(* IEC 61131-3 sources: kerf/packages/kerf-plc/tests/fixtures, 2 files *)

(* ---- blinker.st ---- *)
(* Blinker POU — drives pulse_out at 1 Hz using a TON timer *)
FUNCTION_BLOCK Blinker
VAR
    clock_in : BOOL;
    pulse_out : BOOL;
    t : TON;
END_VAR

(* Update the on-delay timer *)
t(IN := clock_in, PT := T#1s);

(* Latch output from timer Q output *)
pulse_out := t.Q;

END_FUNCTION_BLOCK

(* ---- conveyor.st ---- *)
(* Conveyor POU — start/stop/e-stop control with motor output *)
FUNCTION_BLOCK Conveyor
VAR_INPUT
    start_btn  : BOOL;
    stop_btn   : BOOL;
    estop      : BOOL;
END_VAR
VAR_OUTPUT
    motor_run  : BOOL;
    fault_lamp : BOOL;
END_VAR
VAR
    running    : BOOL;
END_VAR

(* Emergency stop overrides everything *)
IF estop THEN
    running    := FALSE;
    fault_lamp := TRUE;
ELSIF start_btn AND NOT stop_btn THEN
    running    := TRUE;
    fault_lamp := FALSE;
ELSIF stop_btn THEN
    running    := FALSE;
    fault_lamp := FALSE;
ELSE
    fault_lamp := FALSE;
END_IF

motor_run := running;

END_FUNCTION_BLOCK
